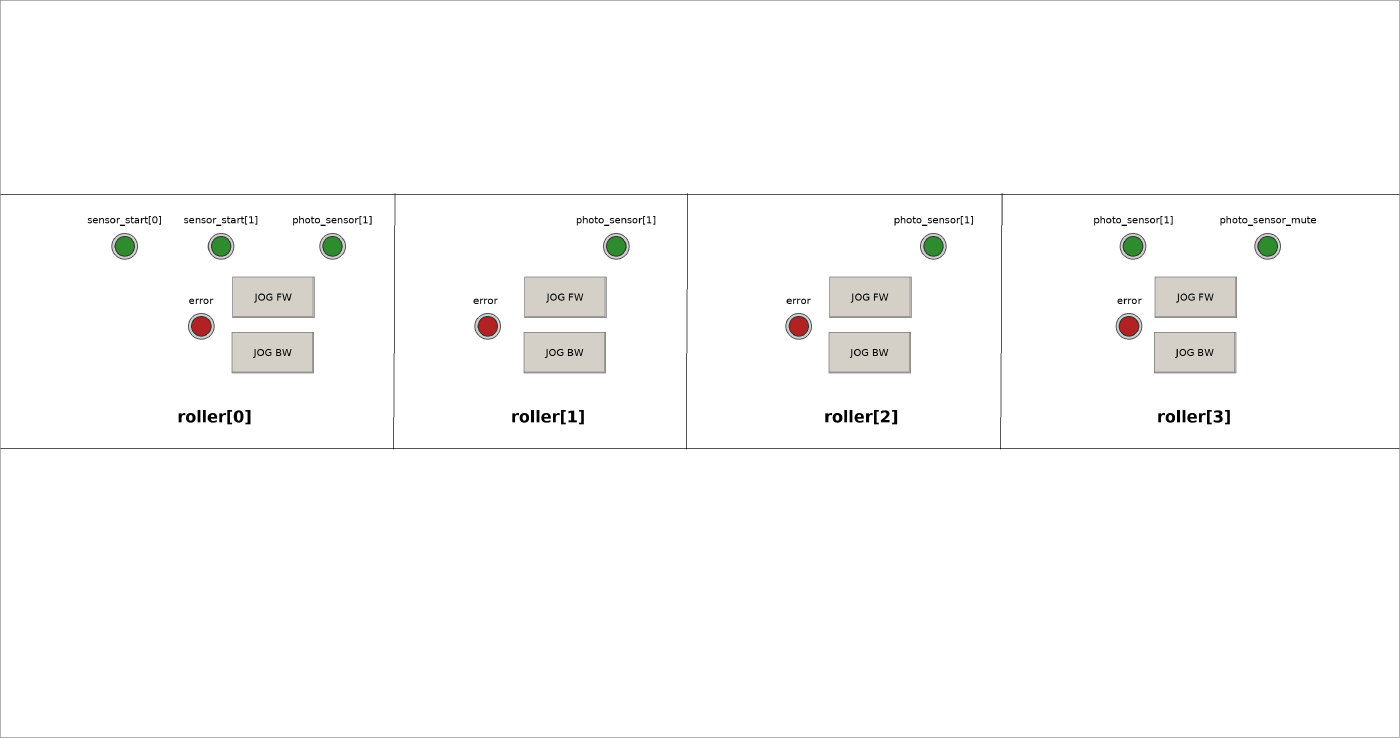
VISUALIZATION v_io_buffer  // 2048x1080
    Lamp1 (464,338 45x45), variable: GVL.fb_buffer.fb_rollers[0].roller.sensor.Q, style: Lamp-Lamp1-Green
    Label (386,309 200x26), "photo_sensor[1]"
    Lamp1 (272,455 45x45), variable: GVL.fb_buffer.fb_rollers[0].roller.err, style: Lamp-Lamp1-Red
    Label (194,427 200x26), "error"
    Label (248,597 132x26), "roller[0]"
    Line (0,284) (2048,284)
    Button (340,405 120x60), "JOG FW", colour toggle: GVL.fb_buffer.fb_rollers[0].roller.forward
        OnMouseDown: execute { GVL.fb_buffer.fb_rollers[0].roller.forward	:= TRUE; }
        OnMouseUp: execute { GVL.fb_buffer.fb_rollers[0].roller.forward	:= FALSE; }
    Button (339,486 120x60), "JOG BW", colour toggle: GVL.fb_buffer.fb_rollers[0].roller.backward
        OnMouseDown: execute { GVL.fb_buffer.fb_rollers[0].roller.backward	:= TRUE; }
        OnMouseUp: execute { GVL.fb_buffer.fb_rollers[0].roller.backward	:= FALSE; }
    Line (0,656) (2048,656)
    Lamp1 (160,338 45x45), variable: GVL.fb_buffer.sensor_start[0].Q, style: Lamp-Lamp1-Green
    Label (82,309 200x26), "sensor_start[0]"
    Lamp1 (879,338 45x45), variable: GVL.fb_buffer.fb_rollers[1].roller.sensor.Q, style: Lamp-Lamp1-Green
    Label (801,309 200x26), "photo_sensor[1]"
    Lamp1 (691,455 45x45), variable: GVL.fb_buffer.fb_rollers[1].roller.err, style: Lamp-Lamp1-Red
    Label (610,427 200x26), "error"
    Label (736,597 132x26), "roller[1]"
    Button (767,405 120x60), "JOG FW", colour toggle: GVL.fb_buffer.fb_rollers[1].roller.forward
        OnMouseDown: execute { GVL.fb_buffer.fb_rollers[1].roller.forward	:= TRUE; }
        OnMouseUp: execute { GVL.fb_buffer.fb_rollers[1].roller.forward	:= FALSE; }
    Button (766,486 120x60), "JOG BW", colour toggle: GVL.fb_buffer.fb_rollers[1].roller.backward
        OnMouseDown: execute { GVL.fb_buffer.fb_rollers[1].roller.backward	:= TRUE; }
        OnMouseUp: execute { GVL.fb_buffer.fb_rollers[1].roller.backward	:= FALSE; }
    Lamp1 (1343,338 45x45), variable: GVL.fb_buffer.fb_rollers[2].roller.sensor.Q, style: Lamp-Lamp1-Green
    Label (1266,309 200x26), "photo_sensor[1]"
    Lamp1 (1146,455 45x45), variable: GVL.fb_buffer.fb_rollers[2].roller.err, style: Lamp-Lamp1-Red
    Label (2867,952 200x26), "error"
    Label (1194,597 132x26), "roller[2]"
    Button (1213,405 120x60), "JOG FW", colour toggle: GVL.fb_buffer.fb_rollers[2].roller.forward
        OnMouseDown: execute { GVL.fb_buffer.fb_rollers[2].roller.forward	:= TRUE; }
        OnMouseUp: execute { GVL.fb_buffer.fb_rollers[2].roller.forward	:= FALSE; }
    Button (1212,486 120x60), "JOG BW", colour toggle: GVL.fb_buffer.fb_rollers[2].roller.backward
        OnMouseDown: execute { GVL.fb_buffer.fb_rollers[2].roller.backward	:= TRUE; }
        OnMouseUp: execute { GVL.fb_buffer.fb_rollers[2].roller.backward	:= FALSE; }
    Lamp1 (1635,338 45x45), variable: GVL.fb_buffer.fb_rollers[3].roller.sensor.Q, style: Lamp-Lamp1-Green
    Label (1558,309 200x26), "photo_sensor[1]"
    Lamp1 (1629,455 45x45), variable: GVL.fb_buffer.fb_rollers[2].roller.err, style: Lamp-Lamp1-Red
    Label (1552,427 200x26), "error"
    Label (1681,597 132x26), "roller[3]"
    Button (1689,405 120x60), "JOG FW", colour toggle: GVL.fb_buffer.fb_rollers[3].roller.forward
        OnMouseDown: execute { GVL.fb_buffer.fb_rollers[3].roller.forward	:= TRUE; }
        OnMouseUp: execute { GVL.fb_buffer.fb_rollers[3].roller.forward	:= FALSE; }
    Button (1688,486 120x60), "JOG BW", colour toggle: GVL.fb_buffer.fb_rollers[3].roller.backward
        OnMouseDown: execute { GVL.fb_buffer.fb_rollers[3].roller.backward	:= TRUE; }
        OnMouseUp: execute { GVL.fb_buffer.fb_rollers[3].roller.backward	:= FALSE; }
    Lamp1 (1832,338 45x45), variable: GVL.fb_buffer.fb_rollers[3].sensor_mute.Q, style: Lamp-Lamp1-Green
    Label (1755,309 200x26), "photo_sensor_mute"
    Lamp1 (301,338 45x45), variable: GVL.fb_buffer.sensor_start[1].Q, style: Lamp-Lamp1-Green
    Label (223,309 200x26), "sensor_start[1]"
    Line (576,657) (578,283)
    Line (1004,657) (1006,283)
    Line (1464,657) (1466,283)
    Label (1068,427 200x26), "error"
END_VISUALIZATION

(* stored: Version 1.1.0.1, ProductVersion 3.1.4024.12
   Visu v_io_buffer: Id {878b60c2-d46b-48ab-bd7d-ad3c48627796} *)
